Staubli VAL3: SAVEJOB.pgx

public program saveJob(num handle_, string value_, bool& result_[])
begin
  // save the current job to given file
  nCommand[handle_]=coTF
  call sendCommand(handle_,"tf"+value_,result_)
end
